{attribute 'linkalways'} 
{attribute 'no_explicit_call' := 'This FB is a CLASS and must be accessed using methods or properties'}
{attribute 'enable_dynamic_creation'}
FUNCTION_BLOCK Node_ContainerType_Vector_TcVnPoint3_LREAL EXTENDS Node
VAR
    out : _GUID;
END_VAR

METHOD PUBLIC  Clone : I_Node
VAR
	pNode : POINTER TO Node_ContainerType_Vector_TcVnPoint3_LREAL;
END_VAR
pNode := __NEW(Node_ContainerType_Vector_TcVnPoint3_LREAL);
Clone := pNode^;
END_METHOD

METHOD FB_init : BOOL
VAR_INPUT
	bInitRetains : BOOL; // if TRUE, the retain variables are initialized (warm start / cold start)
	bInCopyCode : BOOL;  // if TRUE, the instance afterwards gets moved into the copy code (online change)
END_VAR
AddOutput('out', out);
END_METHOD

METHOD PROTECTED OnExecute
out.Value := ContainerType_Vector_TcVnPoint3_LREAL;
END_METHOD

END_FUNCTION_BLOCK

(* stored: Version 1.1.0.1, ProductVersion 3.1.4026.17
   POU Node_ContainerType_Vector_TcVnPoint3_LREAL: Id {698282a3-15c9-0c2f-2b87-26c0cedf579e}, SpecialFunc None
   Folder Constructor: Id {5e057ecf-17dd-0501-1097-9286d8a7ade8}
   Method Clone: Id {56f6aeac-fd17-0398-3f7c-93ac285eb50d}
   Method FB_init: Id {60e84734-f9f8-0ec6-1ea4-1b7e364e67f9}
   Method OnExecute: Id {83b85d33-a224-01f9-345d-34d5bb309cd6} *)
